KUKA KRL program: place_on_playingfield.src, place_on_playingfield.dat

--- place_on_playingfield.src ---
&ACCESS RVO1
&REL 8
&PARAM DISKPATH = KRC:\R1\Program
DEF place_on_playingfield(target:IN)
   DECL FRAME target

   ;FOLD Gripper SET [1]Gripper State=[2]CLOSE Wait 0.2[s] Check with Strategy 1 ;%{PE}
   ;FOLD Parameters Parameters ;%{h}
   ;Params IlfProvider=GripperTech.GripperSet;setgripper=1;setstate=2;setcont=nocont;waittime=0.2;errorstrategy=1
   ;ENDFOLD
   GRPg_SetStateAndCheck(1, 2, 0.2, 1)
   ;ENDFOLD

   $BASE = SBASE(17)
   $TOOL = TOOL_DATA[13]
   $GEAR_JERK[1] = 50.0
   $GEAR_JERK[2] = 50.0
   $GEAR_JERK[3] = 50.0
   $GEAR_JERK[4] = 50.0
   $GEAR_JERK[5] = 50.0
   $GEAR_JERK[6] = 50.0

   target.Z = 100.0
   SPTP target

   target.Z = 0            ; z value of target point is always zero
   $VEL=SVEL_CP(2)
   SLIN target

   GRPg_SetStateAndCheck(1, 1, 0.2, 1)   ; release gripper

   target.Z = 100.0           ; move back to (safe) position above target point
   SLIN target
END

--- place_on_playingfield.dat ---
&ACCESS RVO1
&REL 8
&PARAM DISKPATH = KRC:\R1\Program
DEFDAT  place_on_playingfield PUBLIC
DECL FDAT FP1={TOOL_NO 1,BASE_NO 17,IPO_FRAME #BASE,POINT2[] " ",TQ_STATE FALSE}
DECL PDAT PPDAT1={VEL 100.000,ACC 100.000,APO_DIST 100.000,GEAR_JERK 50.0000,EXAX_IGN 0}
DECL BASIS_SUGG_T LAST_BASIS={POINT1[] "P0                      ",POINT2[] "P0                      ",CP_PARAMS[] "CPDAT0                  ",PTP_PARAMS[] "PDAT0                   ",CONT[] "                        ",CP_VEL[] "2.0                     ",PTP_VEL[] " 100                    ",SYNC_PARAMS[] "SYNCDAT                 ",SPL_NAME[] "S0                      ",A_PARAMS[] "ADAT0                   "}
DECL E6POS XTESTROTATE={X -1.01062298,Y 14.6834211,Z 100.020187,A -2.83435774,B 27.3230839,C -178.171143,S 2,T 34,E1 0.0,E2 0.0,E3 0.0,E4 0.0,E5 0.0,E6 0.0}
DECL FDAT Ftestrotate={TOOL_NO 13,BASE_NO 17,IPO_FRAME #BASE,POINT2[] " ",TQ_STATE FALSE}
DECL PDAT PPDAT2={VEL 100.000,ACC 100.000,APO_DIST 100.000,GEAR_JERK 50.0000,EXAX_IGN 0}
DECL PDAT PPDAT3={VEL 100.000,ACC 100.000,APO_DIST 100.000,GEAR_JERK 50.0000,EXAX_IGN 0}
ENDDAT
